Staubli VAL3: WipeCacheRoom3.pgx

program WipeCacheRoom3()
  local num nNum
begin
  for nNum=1000 to 1499
    sString[nNum]=""
    pfrmCad[nNum].trsf={0,0,0,0,0,0}
  endFor

end
